FUNCTION_BLOCK SludgeBufferActuators (* Composite Function Block Type *)
  (* Standard: 61499-2 *)
  (* Version 0.0, 11/16/2023, SESA371406, Schneider Electric, template *)
  PACKAGE SE.Nereda;
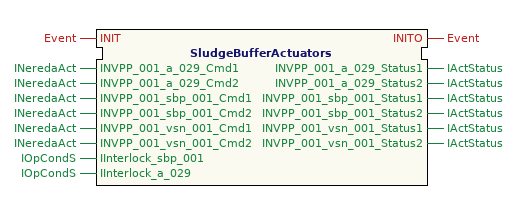
  EVENT_INPUT
    INIT;
  END_EVENT
  EVENT_OUTPUT
    INITO;
  END_EVENT
  SOCKETS
    INVPP_001_a_029_Cmd1 : INeredaAct;
    INVPP_001_a_029_Cmd2 : INeredaAct;
    INVPP_001_sbp_001_Cmd1 : INeredaAct;
    INVPP_001_sbp_001_Cmd2 : INeredaAct;
    INVPP_001_vsn_001_Cmd1 : INeredaAct;
    INVPP_001_vsn_001_Cmd2 : INeredaAct;
    IInterlock_sbp_001 : IOpCondS; (* Condition summary chain input from upstream blocks *)
    IInterlock_a_029 : IOpCondS; (* Condition summary chain input from upstream blocks *)
  END_SOCKETS
  PLUGS
    INVPP_001_a_029_Status1 : IActStatus;
    INVPP_001_a_029_Status2 : IActStatus;
    INVPP_001_sbp_001_Status1 : IActStatus;
    INVPP_001_sbp_001_Status2 : IActStatus;
    INVPP_001_vsn_001_Status1 : IActStatus;
    INVPP_001_vsn_001_Status2 : IActStatus;
  END_PLUGS
  (* 01 - FUNCTIONNAL INPUT INTERFACE *)
  (* 00 - INITIALIZATION *)
  (* 05 - LOGIC *)
  (* 06 - HMI INTERFACE *)
  (* 03 - FIELD INTERFACE *)
  (* 02 - FUNCTIONNAL OUTPUT INTERFACE *)
  (* Actuators Status *)
  (* 04 - CHILDREN *)
  (* 4A - TYPICALS *)
  (* Actuators Command *)
  (* Reset All Actuators *)
  FBS
    ResetAllValves : ResetValvesManager;
    NVPP_001_a_029 : ValveS;
    NVPP_001_a_029_Status : MultiActStatus;
    NVPP_001_sbp_001_Status : MultiActStatus;
    NVPP_001_vsn_001_Status : MultiActStatus;
    NVPP_001_a_029_Cmd : MultiNeredaCmd;
    NVPP_001_sbp_001_Cmd : MultiNeredaCmd;
    NVPP_001_vsn_001_Cmd : MultiNeredaCmd;
    NVPP_001_sbp_001 : Motor_VS;
    NVPP_001_vsn_001 : MotorS;
  END_FBS
  EVENT_CONNECTIONS
    INIT TO ResetAllValves.INIT;
    ResetAllValves.INITO TO INITO;
  END_CONNECTIONS
  ADAPTER_CONNECTIONS
    INVPP_001_a_029_Cmd1 TO NVPP_001_a_029_Cmd.F1CE5E5BC0F88348;
    INVPP_001_a_029_Cmd2 TO NVPP_001_a_029_Cmd.814FBE7646911966;
    INVPP_001_sbp_001_Cmd1 TO NVPP_001_sbp_001_Cmd.F1CE5E5BC0F88348;
    INVPP_001_sbp_001_Cmd2 TO NVPP_001_sbp_001_Cmd.814FBE7646911966;
    INVPP_001_vsn_001_Cmd1 TO NVPP_001_vsn_001_Cmd.F1CE5E5BC0F88348;
    INVPP_001_vsn_001_Cmd2 TO NVPP_001_vsn_001_Cmd.814FBE7646911966;
    IInterlock_sbp_001 TO NVPP_001_sbp_001.9C9EE774F196CD99;
    NVPP_001_a_029_Cmd.30D463C0CF465CCB TO NVPP_001_a_029.476D0447CF6D114C;
    NVPP_001_sbp_001_Cmd.30D463C0CF465CCB TO NVPP_001_sbp_001.D01B7CFFEEA98E7A;
    NVPP_001_vsn_001_Cmd.30D463C0CF465CCB TO NVPP_001_vsn_001.E1DAD7A3AF5C79A5;
    NVPP_001_a_029.E9B1CB906EB3FD07 TO NVPP_001_a_029_Status.18836B5B646921E0;
    NVPP_001_sbp_001.378A5C96F2B54F0C TO NVPP_001_sbp_001_Status.18836B5B646921E0;
    NVPP_001_vsn_001.C98AECEA49DEE5FC TO NVPP_001_vsn_001_Status.18836B5B646921E0;
    ResetAllValves.2 TO NVPP_001_a_029.76FFF418213BE03C;
    NVPP_001_a_029_Status.8244952938F4EC92 TO INVPP_001_a_029_Status1;
    NVPP_001_a_029_Status.3FD61FA75EE1C84B TO INVPP_001_a_029_Status2;
    NVPP_001_sbp_001_Status.8244952938F4EC92 TO INVPP_001_sbp_001_Status1;
    NVPP_001_sbp_001_Status.3FD61FA75EE1C84B TO INVPP_001_sbp_001_Status2;
    NVPP_001_vsn_001_Status.8244952938F4EC92 TO INVPP_001_vsn_001_Status1;
    NVPP_001_vsn_001_Status.3FD61FA75EE1C84B TO INVPP_001_vsn_001_Status2;
    IInterlock_a_029 TO NVPP_001_a_029.9C9EE774F196CD99;
  END_CONNECTIONS
END_FUNCTION_BLOCK
